Staubli VAL3: USERPAGE.pjx

--- USERPAGE.pjx ---
Parameters version=s7.8.3 stackSize=5000 millimeterUnit=true
Program file=changeValue.pgx
Program file=clear.pgx
Program file=divideString.pgx
Program file=editNum.pgx
Program file=editNumField.pgx
Program file=editStr.pgx
Program file=example.pgx
Program file=findPos.pgx
Program file=getListPosition.pgx
Program file=getMenu.pgx
Program file=getNum.pgx
Program file=getView.pgx
Program file=insertDialog.pgx
Program file=isListEmpty.pgx
Program file=leftPos.pgx
Program file=listadd.pgx
Program file=listcreate.pgx
Program file=listcursor.pgx
Program file=listdel.pgx
Program file=listempty.pgx
Program file=listevent.pgx
Program file=listframe.pgx
Program file=listins.pgx
Program file=listredraw.pgx
Program file=listupdate.pgx
Program file=midPos.pgx
Program file=nullKey.pgx
Program file=numCopy.pgx
Program file=printScroll.pgx
Program file=questionDialog.pgx
Program file=read.pgx
Program file=rightPos.pgx
Program file=scroll.pgx
Program file=selectNewField.pgx
Program file=setCenter.pgx
Program file=setList.pgx
Program file=setMenu.pgx
Program file=SetProerty.pgx
Program file=setSizeList.pgx
Program file=setView.pgx
Program file=showBoolStatus.pgx
Program file=strfill.pgx
Program file=strfillchr.pgx
Program file=stringCopy.pgx
Program file=stringToArray.pgx
Program file=strlength.pgx
Program file=timerDialog.pgx
Program file=type.pgx
Program file=typeCenter.pgx
Program file=typeLen.pgx
Program file=typeMenu.pgx
Program file=yes.pgx
Program file=yes_no.pgx
Program file=yes_no_cancel.pgx
Data file=userPage.dtx

--- USERPAGE.dtx ---
bool Show
public bool bListItemRef
bool bReadWrite = true
public bool bShowDialog
public bool bUseEscape
public bool bUseRefresh = true
public num nBottomX[2]
  [0] = 18
  [1] = 18
public num nBottomY = 11
num nFirst
num nKey
num nOffSet
num nOldValue[2]
  [0] = 200
  [1] = 200
public num nPage = 100000
public num nParaAdjustType
num nTest
public num nToSuperV = -1
public num nTopX[2]
  [0] = 20
  [1] = 20
public num nTopY
public num nView
public string sItems = "Name"
string sMessage = "是否删除该项?"
public string sTitle = "工具"
public string sToSuperV
string stest[11]
  [0] = "sbx"
  [1] = "sdfgsd"
  [2] = "bsfghsfh"
  [3] = "sdfgsdfg"
  [4] = "shsgh"
  [5] = "ghdfh"
  [6] = "snsfg"
  [7] = "sfgsg"
  [8] = "sfgsdfg"
  [9] = "sfgs"
  [10] = "dfsgs"
string stest2
string stest3

--- changeValue.pgx ---
public program changeValue(num& x_nValue[] (dimensions=1), num x_nMin (dimensions=1), num x_nMax (dimensions=1), num x_nX (dimensions=1), num x_nY (dimensions=1), string& x_sItems[] (dimensions=1))
  local num l_nOldValue[2]
  local string l_sItem
  local string l_sMessage
  local bool l_bComma
  local string l_sEmpty
begin
  //---------------------------------
  // Staubli copyright 2005
  //                By toneage
  //[Public]-------------------------
  //
  // x_nValue:  num to change
  // x_nMax:    max value
  // x_nMin:    min value
  // x_nX:      X position
  // x_nY:      Y position
  // x_sItems   message
  //
  // look if the value is between max and min
  //
  if x_nMin>x_nMax
    return
  endIf
  //
  // print the line in white
  //
  // call listCleanLine()
  //
  call nullKey(nKey)
  l_nOldValue[1]=round(x_nValue)
  x_nValue=(round(x_nValue*1000))/1000
  l_nOldValue=x_nValue
  // check if is using the comma or not
  if l_nOldValue!=l_nOldValue[1]
    l_bComma=true
  else
    l_bComma=false
  endIf
  // start
  call clear(0,13)
  do
    if x_sItems==""
      //
      //  use the get num
      //
      if l_bComma
        call strfill(l_sEmpty,len(toString(".3",x_nValue)),l_sEmpty)
      else
        call strfill(l_sEmpty,len(toString(".3",x_nValue)),l_sEmpty)
      endIf
      call type(x_nX,x_nY,l_sEmpty)
      gotoxy(x_nX,x_nY)
      nKey=get(x_nValue)
      // check the comma again
      if round(x_nValue)!=x_nValue
        l_bComma=true
      endIf
      //
      // CHECK for MIN MAX VALUE
      //
      if x_nMax!=x_nMin or x_nMin!=0
        if x_nValue>x_nMax
          //
          // ask if you want to continue
          //
          popUpMsg("MAX: "+toString(".2",x_nMax))
          x_nValue=l_nOldValue
          //x_nValue=x_nMax
          nKey=-1
        else
          if x_nValue<x_nMin
            //
            popUpMsg("MIN: "+toString(".2",x_nMin))
            //x_nValue=x_nMin
            x_nValue=l_nOldValue
            nKey=-1
          endIf
        endIf
      endIf
      //
      // UPDATE THE VALUE
      //
      if l_bComma
        call type(x_nX,x_nY,toString(".2",x_nValue))
      else
        call type(x_nX,x_nY,toString("",x_nValue))
      endIf
    else
      // STRING CHOICE
      nKey=getKey()
      switch nKey
        // CHANGE THE ITEMS ARRAY
        case 261
          // UP
          x_nValue=abs((x_nValue+1)%size(x_sItems))
        break
        case 266
          // DOWN
          x_nValue=abs((x_nValue+size(x_sItems)-1)%size(x_sItems))
        break
      endSwitch
      //
      // UPDATE THE VALUE
      //
      setTextMode(3)
      call typeLen(x_nX,x_nY,x_sItems[x_nValue],8)
      setTextMode(0)
    endIf
    // release the resource
    delay(0)
  until nKey==270 or nKey==255
  if nKey==255
    bUseEscape=true
    x_nValue=l_nOldValue
    if x_sItems!=""
      x_sItems=x_sItems[l_nOldValue]
    endIf
  else
    bUseEscape=false
  endIf
  // leave the resource
  delay(0)
end

--- EDITNUM.pgx ---
public program editNum(string& x_sItem, string& x_sItemValue, num& x_nValue, num x_nSelect)
  local string l_sEmpty
  local num l_nValue
  local bool l_bRes
  local num l_nKey
  local num l_nPos
begin
  //
  do
    call clear(0,13)
    call findPos(x_sItem,":",l_nPos)
    gotoxy(nTopX+1,nTopY+nView+1)
    setTextMode(0)
    put(x_sItem)
    call strlength(l_sEmpty,nBottomX-l_nPos+1)
    call type(nTopX+l_nPos+2,nTopY+nView+1,l_sEmpty)
    gotoxy(nTopX+l_nPos+2,nTopY+nView+1)
    toNum(x_sItemValue,l_nValue,l_bRes)
    l_nKey=get(l_nValue)
    if l_nKey==270
      x_sItemValue=toString(".3",l_nValue)
      x_nValue=l_nValue
    endIf
    call strfill(x_sItem,l_nPos+1,x_sItem)
    x_sItem=x_sItem+x_sItemValue
    call strlength(x_sItem,nBottomX+1)
    gotoxy(nTopX+1,nTopY+nView+1)
    setTextMode(1)
    call type(nTopX+1,nTopY+nView+1,x_sItem)
    setTextMode(0)
    delay(0)
  until l_nKey==270 or l_nKey==255

end

--- editNumField.pgx ---
public program editNumField(string x_sTitle, string& x_sItemName[], num& x_nItem[], num& x_nMin[], num& x_nMax[])
  local num j
  local num l_nSize
  local num l_nKey
  local string l_sEvent
  local num l_nIndex
  local num l_nField
  local string l_sItem
  local num i
  local string l_sEmpty[2]
  local string l_sString1
  local num l_nFollow
  local string l_sMsg
begin
  //clear & copy
  nView=nFirst=0
  call listempty()
  call numCopy(x_nItem,nOldValue)
  call numCopy(x_nItem,nOffSet)
  for j=0 to size(nOffSet)-1
    nOffSet[j]=0
  endFor
  // take the size
  l_nSize=size(x_sItemName)-1
  // create the LIST
  call setSizeList(2,max((6-l_nSize/2)-2,2)-2,24,min((l_nSize+1),11))
  call listcreate(x_sTitle)
  //
  // insert items
  //
  if nParaAdjustType==1
    for j=0 to l_nSize
      l_sItem=x_sItemName[j]
      if l_sItem!=""
        if j==9
          call strlength(l_sItem,nBottomX/2)
          if x_nItem[j]==0
            l_sMsg=l_sItem+": "+"关"
            call listadd(l_sMsg)
          else
            l_sMsg=l_sItem+": "+"开"
            call listadd(l_sMsg)
          endIf
        else
          call strlength(l_sItem,nBottomX/2)
          l_sMsg=l_sItem+": "+toString(".4",x_nItem[j])
          call listadd(l_sMsg)
        endIf
        nOffSet[j]=nOffSet[max(j-1,0)]
      else
        nOffSet[j]=nOffSet[max(j-1,0)]+1
      endIf
    endFor
  endIf
  if nParaAdjustType==2
    for j=0 to l_nSize
      l_sItem=x_sItemName[j]
      if l_sItem!=""
        if j==7
          call strlength(l_sItem,nBottomX/2)
          if x_nItem[j]==0
            l_sMsg=l_sItem+": "+"关"
            call listadd(l_sMsg)
          else
            l_sMsg=l_sItem+": "+"开"
            call listadd(l_sMsg)
          endIf
        else
          call strlength(l_sItem,nBottomX/2)
          l_sMsg=l_sItem+": "+toString(".3",x_nItem[j])
          call listadd(l_sMsg)
        endIf
        nOffSet[j]=nOffSet[max(j-1,0)]
      else
        nOffSet[j]=nOffSet[max(j-1,0)]+1
      endIf
    endFor
  endIf
  if nParaAdjustType==3
    for j=0 to l_nSize
      l_sItem=x_sItemName[j]
      if l_sItem!=""
        call strlength(l_sItem,nBottomX/2)
        l_sMsg=l_sItem+": "+toString(".3",x_nItem[j])
        call listadd(l_sMsg)
        nOffSet[j-nOffSet[max(j-1,0)]]=nOffSet[max(j-1,0)]
        nOffSet[j]=nOffSet[max(j-1,0)]
      else
        nOffSet[j]=nOffSet[max(j-1,0)]+1
      endIf
    endFor
  endIf
  if nParaAdjustType==4
    for j=0 to l_nSize
      l_sItem=x_sItemName[j]
      if l_sItem!=""
        if j==10
          call strlength(l_sItem,nBottomX/2)
          if x_nItem[j]==0
            l_sMsg=l_sItem+": "+"直线"
            call listadd(l_sMsg)
          else
            l_sMsg=l_sItem+": "+"圆弧"
            call listadd(l_sMsg)
          endIf
        else
          call strlength(l_sItem,nBottomX/2)
          l_sMsg=l_sItem+": "+toString(".3",x_nItem[j])
          call listadd(l_sMsg)
        endIf
        nOffSet[j]=nOffSet[max(j-1,0)]
      else
        nOffSet[j]=nOffSet[max(j-1,0)]+1
      endIf
    endFor
  endIf


  // update the list
  call listupdate(0)
  do
    call clear(0,13)
    call typeMenu(8,"OK")
    l_nKey=get()
    call listevent(l_nKey,l_nIndex,l_sEvent)
    // use the offset
    i=l_nIndex+nOffSet[max(l_nIndex,0)]
    // on Enter Key
    if nParaAdjustType==1
      if l_nKey==270
        if l_nIndex==9
          call listcursor(l_nIndex,false)
          if size(x_nMin)==size(x_nItem)
            // use min and max
            l_sEmpty[0]="关"
            l_sEmpty[1]="开"
            call changeValue(x_nItem[l_nIndex],x_nMin[l_nIndex],x_nMax[l_nIndex],nTopX+nBottomX/2+3,nView+nTopY+1,l_sEmpty)
          else
            l_sEmpty[0]="关"
            l_sEmpty[1]="开"
            call changeValue(x_nItem[l_nIndex],x_nMin[l_nIndex],x_nMax[l_nIndex],nTopX+nBottomX/2+3,nView+nTopY+1,l_sEmpty)
          endIf
          // UPDATE
          call listdel(l_nIndex)
          l_sItem=x_sItemName[l_nIndex]
          call strlength(l_sItem,nBottomX/2)
          l_sMsg=l_sItem+": "+l_sEmpty[x_nItem[l_nIndex]]
          call listins(l_sMsg,l_nIndex)
          call listupdate(l_nIndex-nView)
        else
          if l_nIndex>nView
            call listcursor(nView,false)
          else
            call listcursor(l_nIndex,false)
          endIf
          if size(x_nMin)==size(x_nItem)
            // use min and max
            l_sEmpty[0]=""
            l_sEmpty[1]=""
            call changeValue(x_nItem[i],x_nMin[i],x_nMax[i],nTopX+nBottomX/2+3,nView+nTopY+1,l_sEmpty)
          else
            call changeValue(x_nItem[i],x_nMin,x_nMax,nTopX+nBottomX/2+3,nView+nTopY+1,l_sEmpty)
          endIf
          // UPDATE
          call listdel(l_nIndex)
          l_sItem=x_sItemName[i]
          call strlength(l_sItem,nBottomX/2)
          l_sMsg=l_sItem+": "+toString(".3",x_nItem[i])
          call listins(l_sMsg,l_nIndex)
          call listupdate(l_nIndex-nView)
        endIf
      endIf
    endIf
    if nParaAdjustType==2
      if l_nKey==270
        if l_nIndex==7
          call listcursor(l_nIndex,false)
          if size(x_nMin)==size(x_nItem)
            // use min and max
            l_sEmpty[0]="关"
            l_sEmpty[1]="开"
            call changeValue(x_nItem[l_nIndex],x_nMin[l_nIndex],x_nMax[l_nIndex],nTopX+nBottomX/2+3,nView+nTopY+1,l_sEmpty)
          else
            l_sEmpty[0]="关"
            l_sEmpty[1]="开"
            call changeValue(x_nItem[l_nIndex],x_nMin[l_nIndex],x_nMax[l_nIndex],nTopX+nBottomX/2+3,nView+nTopY+1,l_sEmpty)
          endIf
          //UPDATE
          call listdel(l_nIndex)
          l_sItem=x_sItemName[l_nIndex]
          call strlength(l_sItem,nBottomX/2)
          l_sMsg=l_sItem+": "+l_sEmpty[x_nItem[l_nIndex]]
          call listins(l_sMsg,l_nIndex)
          call listupdate(l_nIndex-nView)
        else
          if l_nIndex>nView
            call listcursor(nView,false)
          else
            call listcursor(l_nIndex,false)
          endIf
          if size(x_nMin)==size(x_nItem)
            // use min and max
            l_sEmpty[0]=""
            l_sEmpty[1]=""
            call changeValue(x_nItem[i],x_nMin[i],x_nMax[i],nTopX+nBottomX/2+3,nView+nTopY+1,l_sEmpty)
          else
            call changeValue(x_nItem[i],x_nMin,x_nMax,nTopX+nBottomX/2+3,nView+nTopY+1,l_sEmpty)
          endIf
          // UPDATE
          call listdel(l_nIndex)
          l_sItem=x_sItemName[i]
          call strlength(l_sItem,nBottomX/2)
          l_sMsg=l_sItem+": "+toString(".3",x_nItem[i])
          call listins(l_sMsg,l_nIndex)
          call listupdate(l_nIndex-nView)
        endIf
      endIf
    endIf
    if nParaAdjustType==3
      if l_nKey==270
        if l_nIndex>nView
          call listcursor(nView,false)
        else
          call listcursor(l_nIndex,false)
        endIf
        if size(x_nMin)==size(x_nItem)
          // use min and max
          l_sEmpty[0]=""
          l_sEmpty[1]=""
          call changeValue(x_nItem[i],x_nMin[i],x_nMax[i],nTopX+nBottomX/2+3,nView+nTopY+1,l_sEmpty)
        else
          call changeValue(x_nItem[i],x_nMin,x_nMax,nTopX+nBottomX/2+3,nView+nTopY+1,l_sEmpty)

        endIf
        // UPDATE
        call listdel(l_nIndex)
        l_sItem=x_sItemName[i]
        call strlength(l_sItem,nBottomX/2)
        l_sMsg=l_sItem+": "+toString(".3",x_nItem[i])
        call listins(l_sMsg,l_nIndex)
        call listupdate(l_nIndex-nView)
        //      endIf
      endIf
    endIf
    if nParaAdjustType==4
      if l_nKey==270
        if l_nIndex==9
          call listcursor(l_nIndex,false)
          if size(x_nMin)==size(x_nItem)
            // use min and max
            l_sEmpty[0]="直线"
            l_sEmpty[1]="圆弧"
            call changeValue(x_nItem[l_nIndex],x_nMin[l_nIndex],x_nMax[l_nIndex],nTopX+nBottomX/2+3,nView+nTopY+1,l_sEmpty)
          else
            l_sEmpty[0]="直线"
            l_sEmpty[1]="圆弧"
            call changeValue(x_nItem[l_nIndex],x_nMin[l_nIndex],x_nMax[l_nIndex],nTopX+nBottomX/2+3,nView+nTopY+1,l_sEmpty)
          endIf
          // UPDATE
          call listdel(l_nIndex)
          l_sItem=x_sItemName[l_nIndex]
          call strlength(l_sItem,nBottomX/2)
          l_sMsg=l_sItem+": "+l_sEmpty[x_nItem[l_nIndex]]
          call listins(l_sMsg,l_nIndex)
          call listupdate(l_nIndex-nView)
        else
          if l_nIndex>nView
            call listcursor(nView,false)
          else
            call listcursor(l_nIndex,false)
          endIf
          if size(x_nMin)==size(x_nItem)
            // use min and max
            l_sEmpty[0]=""
            l_sEmpty[1]=""
            call changeValue(x_nItem[i],x_nMin[i],x_nMax[i],nTopX+nBottomX/2+3,nView+nTopY+1,l_sEmpty)
          else
            call changeValue(x_nItem[i],x_nMin,x_nMax,nTopX+nBottomX/2+3,nView+nTopY+1,l_sEmpty)
          endIf
          // UPDATE
          call listdel(l_nIndex)
          l_sItem=x_sItemName[i]
          call strlength(l_sItem,nBottomX/2)
          l_sMsg=l_sItem+": "+toString(".3",x_nItem[i])
          call listins(l_sMsg,l_nIndex)
          call listupdate(l_nIndex-nView)
        endIf
      endIf
    endIf
    delay(0)
  until l_nKey==278 or l_nKey==255
  // escape use????
  if l_nKey==255
    bUseEscape=true
    call numCopy(nOldValue,x_nItem)
  else
    bUseEscape=false
  endIf
  // exit
  call nullKey(l_nKey)
end

--- EDITSTR.pgx ---
public program editStr(string& x_sItem, string& x_sItemValue, num x_nSelect)
  local string l_sEmpty
  local num l_nKey
  local num l_nPos
begin
  //
  do
    call clear(0,13)
    call findPos(x_sItem,":",l_nPos)
    gotoxy(nTopX+1,nTopY+x_nSelect+1)
    setTextMode(0)
    put(x_sItem)
    call strlength(l_sEmpty,nBottomX-l_nPos+1)
    call type(nTopX+l_nPos+2,nTopY+x_nSelect+1,l_sEmpty)
    gotoxy(nTopX+l_nPos+2,nTopY+x_nSelect+1)
    l_nKey=get(x_sItemValue)
    call strfill(x_sItem,l_nPos+1,x_sItem)
    x_sItem=x_sItem+x_sItemValue
    call strlength(x_sItem,nBottomX+1)
    gotoxy(nTopX+1,nTopY+x_nSelect+1)
    setTextMode(1)
    call type(nTopX+1,nTopY+x_nSelect+1,x_sItem)
    setTextMode(0)
    delay(0)
  until l_nKey==270 or l_nKey==255
end

--- getNum.pgx ---
public program getNum(string x_sTitle, num& x_nValue, num x_nMin, num x_nMax)
  local string l_sItemName
  local num l_nKey
  local num l_i
  local num l_nPos
  local num l_nValue
begin
  //获取一个数值
  l_nValue=x_nValue
  do
    call listframe(x_sTitle,10,5,20,1)
    call clear(11,6)
    gotoxy(15,6)
    l_nKey=get(l_nValue)
    //超出范围
    if l_nValue<x_nMin or l_nValue>x_nMax
      popUpMsg("取值范围:"+"["+toString(".3",x_nMin)+","+toString(".3",x_nMax)+"]")
      l_nValue=x_nValue
    else
      x_nValue=l_nValue
    endIf
    delay(0)
  until l_nKey==255

end

--- insertDialog.pgx ---
public program insertDialog(string x_sMsg, num& x_nItem[], num x_nMin, num x_nMax)
  local num l_nStartLine
  local num l_nLine
  local num i
  local num l_nPX
  local num l_nPY
  local string l_sItem
  local string l_sMessage
  local string l_sEmpty
  local string l_sTemp
begin
  //
  // modify the x_sItem, using a min max range
  //
  if watch(bShowDialog==false,2)==false
    bShowDialog=false
    logMsg("error dialog resoursing")
    return
  else
    setMutex(bShowDialog)
    // clear the line
    call clear(0,13)
    // look for the comma
    if round(x_nItem)!=x_nItem
      l_sItem=toString(".2",x_nItem)
    else
      l_sItem=toString("",x_nItem)
    endIf
    // print the line
    l_sTemp=x_sMsg+">"+l_sItem
    call stringCopy(l_sTemp,sMessage)
    // divide the sentence
    call divideString(sMessage,l_nLine)
    l_nStartLine=round(5-l_nLine/2)
    // Start LINE
    call type(0,l_nStartLine-2,"┌──────────────────────────────────────┐")
    call type(0,l_nStartLine-1,"│                                      │")
    // write the message
    for i=0 to l_nLine
      //call type(,"                                      ")
      l_sMessage=sMessage[i]
      call typeCenter(i+l_nStartLine,l_sMessage,38,false)
      call type(0,l_nStartLine+i,"│"+l_sMessage+"│")
    endFor
    // end LINE
    call type(0,l_nStartLine+l_nLine+1,"│                                      │")
    call type(0,l_nStartLine+l_nLine+2,"└──────────────────────────────────────┘")
    l_nPX=find(l_sMessage,">")+2
    l_nPY=l_nStartLine+l_nLine
    // change the value
    call changeValue(x_nItem,x_nMin,x_nMax,l_nPX,l_nPY,l_sEmpty)
    //
    bShowDialog=false
    bUseRefresh=true
    //
    delay(0)
  endIf
end

--- listevent.pgx ---
public program listevent(num pkey (dimensions=1), num& pIndex[] (dimensions=1), string& pItem[] (dimensions=1))
  local num lVal
  local num l_nSize
  local bool l_bEmpty
begin
  //
  // Toneage Staubli product
  //
  //
  // get the item in the list and scroll it
  //

  call isListEmpty(l_bEmpty)
  if !l_bEmpty
    l_nSize=size(sItems)-1
    // check the overFlow
    l_nSize=size(sItems)-1
    if (nFirst+nView>l_nSize)
      // reset the value
      nFirst=nView=0
    endIf
    // security...
    switch (pkey)
      //Up
      case 261
        if ((nView-1)>=0)
          // no need to scroll only change cursor position
          call listcursor(nView,false)
          nView=nView-1
          call listcursor(nView,true)
          // print the scroll
          //call printScroll()
        else
          if nView==0
            // scroll up
            if ((nFirst-1)>=0)
              nFirst=nFirst-1
              call listupdate(nFirst)
            else
              // go to the end
              if nView+nFirst!=l_nSize
                call listcursor(nView,false)
                call selectNewField(l_nSize,nFirst+nView,nView)
              endIf
            endIf
          endIf
        endIf
      break
      //Down
      case 266
        if ((nView+nFirst+1)<size(sItems))
          // no need to scroll only chenge cursor position
          if ((nView+1)<nBottomY)
            call listcursor(nView,false)
            nView=nView+1
            call listcursor(nView,true)
            // print the scroll
            //call printScroll()
          else
            // move UP
            nFirst=nFirst+1
            call listupdate(nFirst)
          endIf
        else
          // go to the top
          if !(nView==0 and nFirst==0)
            call listcursor(nView,false)
            nView=0
            call listupdate(0)
          endIf
        endIf
      break
      //Page Up
      case 262
        if !(nView==0 and nFirst==0)
          call listcursor(nView,false)
          if ((nFirst+nView-nBottomY)>=0)
            // move one page up
            call selectNewField(nFirst+nView-nBottomY,nFirst+nView,nView)
          else
            // go to home
            nView=0
            call listupdate(0)
          endIf
        endIf
      break
      //Page Down
      case 267
        if nView+nFirst!=l_nSize
          call listcursor(nView,false)
          if ((nView+nFirst+nBottomY)<size(sItems)-1)
            // move one page down
            call selectNewField(nFirst+nView+nBottomY,nFirst+nView,nView)
          else
            // go to the end
            call selectNewField(l_nSize,nFirst+nView,nView)
          endIf
        endIf
      break
      //End
      case 269
        if nView+nFirst!=l_nSize
          // move to end
          call listcursor(nView,false)
          call selectNewField(l_nSize,nFirst+nView,nView)
        endIf
      break
      //Home
      case 265
        if !(nView==0 and nFirst==0)
          // move to home
          call listcursor(nView,false)
          nView=0
          call listupdate(0)
        endIf
      break
      default
      break
    endSwitch
    pIndex=nFirst+nView
    pItem=sItems[pIndex]
    //
  else
    // reset the item
    pItem=""
    pIndex=0
  endIf
end

--- printScroll.pgx ---
program printScroll()
  local num i
  local num lX
  local num lY
begin
  //
  // put the scroll
  //
  if size(sItems)>nBottomY
    // find the percentage
    //windows style
    //i=(size(sItems)-nBottomY+1)/(nFirst+1)
    // nokia style
    i=(size(sItems))/(nFirst+nView+1)
    lX=nTopX+nBottomX+1
    lY=roundUp((nBottomY)/i+nTopY)
    for i=nTopY+1 to nBottomY
      gotoxy(lX,i)
      if i==lY
        //
        put("■")
        //
        //    else
        //      put("│")
      endIf
    endFor
  endIf
end

--- SETLIST.pgx ---
public program setList(string x_sTitle, string& x_sListItem[], bool x_bUserRefresh, bool x_bListItemRef, num& x_nSelected, string& x_sItem, num& x_nKey)
  local num l_nView
  local num l_nItem
begin
  if x_bUserRefresh
    if x_bListItemRef
      call setSizeList(20,0,18,11)
      call listcreate(x_sTitle)
      if x_sListItem[0]!=""
        call listadd(x_sListItem)
      endIf
    else
      call setSizeList(20,0,18,11)
      call listframe(x_sTitle,nTopX,nTopY,nBottomX,nBottomY)
    endIf
    call selectNewField(x_nSelected,l_nItem,l_nView)
  endIf
  x_nKey=getKey()
  if x_nKey!=-1
    call listevent(x_nKey,l_nItem,x_sItem)
    l_nView=nView
    x_nSelected=l_nItem
  endIf
end

--- SetProerty.pgx ---
public program SetProerty(string x_sTitle, num x_nTopX, num x_nTopY, num x_nBottomX, num x_nBottomY, string& x_sListItem[], string& x_sItem)
  local num l_nKey
  local num l_nItem
  local string l_sTemp
begin
  call setSizeList(x_nTopX,x_nTopY,x_nBottomX,x_nBottomY)
  call listcreate(x_sTitle)
  call listadd(x_sListItem)
  call listupdate(0)
  call clear(0,13)
  call typeMenu(1,"OK")
  l_sTemp=x_sItem
  do
    l_nKey=getKey()
    call listevent(l_nKey,l_nItem,x_sItem)
    delay(0)
  until l_nKey==271 or l_nKey==255 or l_nKey==270
  if l_nKey==255
    x_sItem=l_sTemp
  endIf
  wait(getKey()==-1)
end

--- YES_NO.PGX ---
public program yes_no(string x_sMessage, string& x_sYesNo[], bool& x_bResult[])
  local num i
  local string l_sButton[2]
begin
  //
  // write a yes no question dialog
  //
  if x_sYesNo!=""
    l_sButton[0]=x_sYesNo
  else
    l_sButton[0]="Yes"
  endIf
  //
  if x_sYesNo[1]!=""
    l_sButton[1]=x_sYesNo[1]
  else
    l_sButton[1]="No"
  endIf
  // question Dialog
  call questionDialog(x_sMessage,l_sButton,i)
  // press F8->YES or ENTER
  if i==1 or i==0
    x_bResult=true
  else
    // press escape or F7->NO
    x_bResult=false
  endIf
end
